PROGRAM MAIN
VAR
	fb_rpc : FB_RPC;
END_VAR

END_PROGRAM

(* stored: Version 1.1.0.1, ProductVersion 3.1.4024.12
   POU MAIN: Id {f874d754-4343-477a-8a97-97d3f1f4f9c7}, SpecialFunc None *)
